// TIA Portal V15.1 export
// export: Created 2024-06-21T08:40:41.6810259Z, ExportSetting WithDefaults, DisplayName Totally Integrated Automation Portal, DisplayVersion V15.1 Update 5, DisplayName TIA Portal Openness, DisplayVersion V15.1 Update 5, DisplayName SINAMICS Startdrive Advanced, DisplayVersion V15.1, DisplayName G130, G150, S120, S150, SINAMICS MV, S210, DisplayVersion V15.1, DisplayName G110M, G120, G120C, G120D, G120P, DisplayVersion V15.1, DisplayName STEP 7 Professional, DisplayVersion V15.1 Update 5, DisplayName STEP 7 Safety, DisplayVersion V15.1, DisplayName WinCC Professional, DisplayVersion V15.1 Update 5, DisplayName SIMATIC Visualization Architect, DisplayVersion V15.1
DATA_BLOCK "_209000NCP01AK"   // DB254
{ S7_Optimized_Access := 'FALSE' }
AUTHOR : VCC
NAME : LocFnc
VERSION : 0.1
// stored: AutoNumber false, DBAccessibleFromOPCUA true, IsOnlyStoredInLoadMemory false, IsWriteProtectedInAS false
   VAR RETAIN
      AA_AK01E1QM1 { ExternalAccessible := 'False'; ExternalVisible := 'False'; ExternalWritable := 'False'} : Bool;   // AE01 EG1 - Overload protection power supply 24VDC
      AA_AK01E1QM4 { ExternalAccessible := 'False'; ExternalVisible := 'False'; ExternalWritable := 'False'} : Bool;   // AK02 EG2 - Overload protection power supply 24VDC
      AA_AK02E3EG2 { ExternalAccessible := 'False'; ExternalVisible := 'False'; ExternalWritable := 'False'} : Bool;   // AK02 EG2 - Power supply 24VDC NOK
      AD_AK02E3FV2 { ExternalAccessible := 'False'; ExternalVisible := 'False'; ExternalWritable := 'False'} : Bool;   // AK02 EG2 - Surge protection 24VDC NOK
      AA_AK02E3FS50_CH1 { ExternalAccessible := 'False'; ExternalVisible := 'False'; ExternalWritable := 'False'} : Bool;   // 24VDC Fuse - General - IO card PLC AE01
      AD_AK02E3FS50_CH2 { ExternalAccessible := 'False'; ExternalVisible := 'False'; ExternalWritable := 'False'} : Bool;   // 24VDC Fuse - General - Doorcontacts
      AA_AK02E3FS51_CH1 { ExternalAccessible := 'False'; ExternalVisible := 'False'; ExternalWritable := 'False'} : Bool;   // 24VDC Fuse - General - DI/DO AK01
      AA_AK02E3FS51_CH2 { ExternalAccessible := 'False'; ExternalVisible := 'False'; ExternalWritable := 'False'} : Bool;   // 24VDC Fuse - General - F-DI/F-DO AK01
      AA_AK02E3FS52_CH1 { ExternalAccessible := 'False'; ExternalVisible := 'False'; ExternalWritable := 'False'} : Bool;   // 24VDC Fuse - General - DI/DO AK03
      AA_AK02E3FS52_CH2 { ExternalAccessible := 'False'; ExternalVisible := 'False'; ExternalWritable := 'False'} : Bool;   // 24VDC Fuse - General - F-DI/F-DO AK03
      AA_AK02E3FS53_CH1 { ExternalAccessible := 'False'; ExternalVisible := 'False'; ExternalWritable := 'False'} : Bool;   // 24VDC Fuse - General - DI/DO AK04
      AA_AK02E3FS53_CH2 { ExternalAccessible := 'False'; ExternalVisible := 'False'; ExternalWritable := 'False'} : Bool;   // 24VDC Fuse - General - F-DI/F-DO AK04
      AA_AK02E3FS54_CH1 { ExternalAccessible := 'False'; ExternalVisible := 'False'; ExternalWritable := 'False'} : Bool;   // 24VDC Fuse - General - DI/DO General Field
      AA_AK02E3FS54_CH2 { ExternalAccessible := 'False'; ExternalVisible := 'False'; ExternalWritable := 'False'} : Bool;   // 24VDC Fuse - General - F-DI/F-DO General Field
      AD_AK02E3FS50_CH1 { ExternalAccessible := 'False'; ExternalVisible := 'False'; ExternalWritable := 'False'} : Bool;   // 24VDC Fuse - General - IO card PLC AE01
      AD_AK02E3FS51_CH1 { ExternalAccessible := 'False'; ExternalVisible := 'False'; ExternalWritable := 'False'} : Bool;   // 24VDC Fuse - General - DI/DO AK01
      AD_AK02E3FS51_CH2 { ExternalAccessible := 'False'; ExternalVisible := 'False'; ExternalWritable := 'False'} : Bool;   // 24VDC Fuse - General - F-DI/F-DO AK01
      AD_AK02E3FS52_CH1 { ExternalAccessible := 'False'; ExternalVisible := 'False'; ExternalWritable := 'False'} : Bool;   // 24VDC Fuse - General - DI/DO AK03
      AD_AK02E3FS52_CH2 { ExternalAccessible := 'False'; ExternalVisible := 'False'; ExternalWritable := 'False'} : Bool;   // 24VDC Fuse - General - F-DI/F-DO AK03
      AD_AK02E3FS53_CH1 { ExternalAccessible := 'False'; ExternalVisible := 'False'; ExternalWritable := 'False'} : Bool;   // 24VDC Fuse - General - DI/DO AK04
      AD_AK02E3FS53_CH2 { ExternalAccessible := 'False'; ExternalVisible := 'False'; ExternalWritable := 'False'} : Bool;   // 24VDC Fuse - General - F-DI/F-DO AK04
      AD_AK02E3FS54_CH1 { ExternalAccessible := 'False'; ExternalVisible := 'False'; ExternalWritable := 'False'} : Bool;   // 24VDC Fuse - General - DI/DO General Field
      AD_AK02E3FS54_CH2 { ExternalAccessible := 'False'; ExternalVisible := 'False'; ExternalWritable := 'False'} : Bool;   // 24VDC Fuse - General - F-DI/F-DO General Field
      AC_AK01E1QM6 { ExternalAccessible := 'False'; ExternalVisible := 'False'; ExternalWritable := 'False'} : Bool;   // 400VAC - Overload protection Cooling unit AK03
      AA_AK01E2FS1 { ExternalAccessible := 'False'; ExternalVisible := 'False'; ExternalWritable := 'False'} : Bool;   // 230VAC - Overload protection 230V AK01
      AC_AK01E2FS2 { ExternalAccessible := 'False'; ExternalVisible := 'False'; ExternalWritable := 'False'} : Bool;   // 230VAC - Overload protection 230V power monitor AK01
      AC_AK01E2FS3 { ExternalAccessible := 'False'; ExternalVisible := 'False'; ExternalWritable := 'False'} : Bool;   // 230VAC - Overload protection Socket + Light AK01-04
      AC_AK01E2FS4 { ExternalAccessible := 'False'; ExternalVisible := 'False'; ExternalWritable := 'False'} : Bool;   // 230VAC - Overload protection Socket + Light AE01-02
      AC_AK01E2FS5 { ExternalAccessible := 'False'; ExternalVisible := 'False'; ExternalWritable := 'False'} : Bool;   // 230VAC - Overload protection Cooling AE01-02
      AC_AK01E2FS6 { ExternalAccessible := 'False'; ExternalVisible := 'False'; ExternalWritable := 'False'} : Bool;   // 230VAC - Overload protection Socket AS01
      AC_AK01E2FS7 { ExternalAccessible := 'False'; ExternalVisible := 'False'; ExternalWritable := 'False'} : Bool;   // 230VAC - Overload protection Socket AS02
      AC_AK03EL1 { ExternalAccessible := 'False'; ExternalVisible := 'False'; ExternalWritable := 'False'} : Bool;   // Fault cooling unit cabinet AK03
      AD_AK01E2SG1 { ExternalAccessible := 'False'; ExternalVisible := 'False'; ExternalWritable := 'False'} : Bool;   // Door not closed cabinet AK01
      AD_AK02E2SG1 { ExternalAccessible := 'False'; ExternalVisible := 'False'; ExternalWritable := 'False'} : Bool;   // Door not closed cabinet AK02
      AD_AK03E2SG1 { ExternalAccessible := 'False'; ExternalVisible := 'False'; ExternalWritable := 'False'} : Bool;   // Door not closed cabinet AK03
      AD_AK04E2SG1 { ExternalAccessible := 'False'; ExternalVisible := 'False'; ExternalWritable := 'False'} : Bool;   // Door not closed cabinet AK04
      AC_AK01QC1 { ExternalAccessible := 'False'; ExternalVisible := 'False'; ExternalWritable := 'False'} : Bool;   // Contactor summary door closed not ok, cabinet AK01-AK02-AK03-AK04
      AD_AK01E1FV1 { ExternalAccessible := 'False'; ExternalVisible := 'False'; ExternalWritable := 'False'} : Bool;   // Surge protection 400VAC AK01 NOK
      AD_AK01E2FV1 { ExternalAccessible := 'False'; ExternalVisible := 'False'; ExternalWritable := 'False'} : Bool;   // Surge protection 230VAC AK01 NOK
      AK01E1QM1AlarmABCondition { ExternalAccessible := 'False'; ExternalVisible := 'False'; ExternalWritable := 'False'} : Bool;   // Alarm AB condition
      AK01E1QM4AlarmABCondition { ExternalAccessible := 'False'; ExternalVisible := 'False'; ExternalWritable := 'False'} : Bool;   // Alarm AB condition
      AK02E3EG2AlarmABCondition { ExternalAccessible := 'False'; ExternalVisible := 'False'; ExternalWritable := 'False'} : Bool;   // Alarm AB condition
      AK02E3FS50_CH1AlarmABCondition { ExternalAccessible := 'False'; ExternalVisible := 'False'; ExternalWritable := 'False'} : Bool;   // Alarm AB condition
      AK02E3FS51_CH1AlarmABCondition { ExternalAccessible := 'False'; ExternalVisible := 'False'; ExternalWritable := 'False'} : Bool;   // Alarm AB condition
      AK02E3FS51_CH2AlarmABCondition { ExternalAccessible := 'False'; ExternalVisible := 'False'; ExternalWritable := 'False'} : Bool;   // Alarm AB condition
      AK02E3FS52_CH1AlarmABCondition { ExternalAccessible := 'False'; ExternalVisible := 'False'; ExternalWritable := 'False'} : Bool;   // Alarm AB condition
      AK02E3FS52_CH2AlarmABCondition { ExternalAccessible := 'False'; ExternalVisible := 'False'; ExternalWritable := 'False'} : Bool;   // Alarm AB condition
      AK02E3FS53_CH1AlarmABCondition { ExternalAccessible := 'False'; ExternalVisible := 'False'; ExternalWritable := 'False'} : Bool;   // Alarm AB condition
      AK02E3FS53_CH2AlarmABCondition { ExternalAccessible := 'False'; ExternalVisible := 'False'; ExternalWritable := 'False'} : Bool;   // Alarm AB condition
      AK02E3FS54_CH1AlarmABCondition { ExternalAccessible := 'False'; ExternalVisible := 'False'; ExternalWritable := 'False'} : Bool;   // Alarm AB condition
      AK02E3FS54_CH2AlarmABCondition { ExternalAccessible := 'False'; ExternalVisible := 'False'; ExternalWritable := 'False'} : Bool;   // Alarm AB condition
      AK01E2FS1AlarmABCondition { ExternalAccessible := 'False'; ExternalVisible := 'False'; ExternalWritable := 'False'} : Bool;   // Alarm AB condition
      H_209000AK01E1QM1IAnim : Word;   // HMI Animation of the icon
      H_209000AK01E1QM4IAnim : Word;   // HMI Animation of the icon
      H_209000AK02E3EG2IAnim : Word;   // HMI Animation of the icon
      H_209000AK02E3FV2IAnim : Word;   // HMI Animation of the icon
      H_209000AK02E3FS50_CH1IAnim : Word;   // HMI Animation of the icon
      H_209000AK02E3FS50_CH2IAnim : Word;   // HMI Animation of the icon
      H_209000AK02E3FS51_CH1IAnim : Word;   // HMI Animation of the icon
      H_209000AK02E3FS51_CH2IAnim : Word;   // HMI Animation of the icon
      H_209000AK02E3FS52_CH1IAnim : Word;   // HMI Animation of the icon
      H_209000AK02E3FS52_CH2IAnim : Word;   // HMI Animation of the icon
      H_209000AK02E3FS53_CH1IAnim : Word;   // HMI Animation of the icon
      H_209000AK02E3FS53_CH2IAnim : Word;   // HMI Animation of the icon
      H_209000AK02E3FS54_CH1IAnim : Word;   // HMI Animation of the icon
      H_209000AK02E3FS54_CH2IAnim : Word;   // HMI Animation of the icon
      H_209000AK02E3FS55_CH2IAnim : Word;   // HMI Animation of the icon
      H_209000AK02E3FS56_CH2IAnim : Word;   // HMI Animation of the icon
      H_209000AK02E3FS57_CH1IAnim : Word;   // HMI Animation of the icon
      H_209000AK02E3FS57_CH2IAnim : Word;   // HMI Animation of the icon
      H_209000AK01E1QM6IAnim : Word;   // HMI Animation of the icon
      H_209000AK01E2FS1IAnim : Word;   // HMI Animation of the icon
      H_209000AK01E2FS2IAnim : Word;   // HMI Animation of the icon
      H_209000AK01E2FS3IAnim : Word;   // HMI Animation of the icon
      H_209000AK01E2FS4IAnim : Word;   // HMI Animation of the icon
      H_209000AK01E2FS5IAnim : Word;   // HMI Animation of the icon
      H_209000AK01E2FS6IAnim : Word;   // HMI Animation of the icon
      H_209000AK01E2FS7IAnim : Word;   // HMI Animation of the icon
      H_209000AK03EL1IAnim : Word;   // HMI Animation of the icon
      H_209000AK01E2SG1IAnim : Word;   // HMI Animation of the icon
      H_209000AK02E2SG1IAnim : Word;   // HMI Animation of the icon
      H_209000AK03E2SG1IAnim : Word;   // HMI Animation of the icon
      H_209000AK04E2SG1IAnim : Word;   // HMI Animation of the icon
      H_209000AK01QC1IAnim : Word;   // HMI Animation of the icon
      H_209000AK01E1FV1IAnim : Word;   // HMI Animation of the icon
      H_209000AK01E2FV1IAnim : Word;   // HMI Animation of the icon
      H_DBnr : Int;   // DB number
      H_Anim : Word;   // Animation
      H_HMI : Struct   // Icon Animation
         "209000AK02JC32" : "H_HMI";   // HMI Animation of the icon
      END_STRUCT;
      H : Struct   // Animation
         "209000AK02JC32" : "H_ETAFuseCPC20PN";   // HMI Animation
      END_STRUCT;
      H_LoccBoxGlobalSignals : Struct   // Global signals between all the FB's
         Busy : Bool;   // Busy with GET the info from one of the fuses
         DBnrFromPopup : Int;   // The return DB number from the pop-up that is open
      END_STRUCT;
      AlarmA { ExternalAccessible := 'False'; ExternalVisible := 'False'; ExternalWritable := 'False'} : Bool;   // Alarm A
      AlarmB { ExternalAccessible := 'False'; ExternalVisible := 'False'; ExternalWritable := 'False'} : Bool;   // Alarm B
      AlarmC { ExternalAccessible := 'False'; ExternalVisible := 'False'; ExternalWritable := 'False'} : Bool;   // Alarm C
      AlarmD { ExternalAccessible := 'False'; ExternalVisible := 'False'; ExternalWritable := 'False'} : Bool;   // Alarm D
      AlarmABCondition { ExternalAccessible := 'False'; ExternalVisible := 'False'; ExternalWritable := 'False'} : Bool;   // Alarm AB condition
      "AK02-JC32" { ExternalAccessible := 'False'; ExternalVisible := 'False'; ExternalWritable := 'False'} : "AlarmBits";   // ETA fuse Alarm Bits
      "AK02-JC32_ETAFuseData" { ExternalAccessible := 'False'; ExternalVisible := 'False'; ExternalWritable := 'False'} : "ETAFuseData";   // ETA fuse status
   END_VAR
BEGIN
END_DATA_BLOCK
